{attribute 'linkalways'} 
{attribute 'no_explicit_call' := 'This FB is a CLASS and must be accessed using methods or properties'}
{attribute 'enable_dynamic_creation'}
FUNCTION_BLOCK FINAL LE_LREAL EXTENDS Node
VAR
	in1 : _LREAL(0.0);
	in2 : _LREAL(0.0);
	out : _BOOL(FALSE);
END_VAR

METHOD PUBLIC Clone : I_Node
VAR
	pNode : POINTER TO LE_LREAL;
END_VAR
pNode := __NEW(LE_LREAL);
Clone := pNode^;
END_METHOD

METHOD FB_init : BOOL
VAR_INPUT
	bInitRetains : BOOL; // if TRUE, the retain variables are initialized (warm start / cold start)
	bInCopyCode : BOOL;  // if TRUE, the instance afterwards gets moved into the copy code (online change)
END_VAR
AddInput('in1',THIS^.in1);
AddInput('in2',THIS^.in2);
AddOutput('out', THIS^.out);
END_METHOD

METHOD PROTECTED OnExecute
VAR
END_VAR
out.Value := in1.Value <= in2.Value;
END_METHOD

END_FUNCTION_BLOCK

(* stored: Version 1.1.0.1, ProductVersion 3.1.4024.15
   POU LE_LREAL: Id {a046585e-4c3f-48a1-aa94-604d72e406f2}, SpecialFunc None
   Folder Constructor: Id {fc5c9e07-ebd8-4389-9a38-f342f986f6d8}
   Method Clone: Id {746db0e6-5e02-4256-9f9e-eb18471f30d8}
   Method FB_init: Id {178d8a11-8222-43ff-b204-8fbbf966067b}
   Method OnExecute: Id {9e47d0c5-ce06-4636-a15a-f1c1a9f1e70d} *)
